(* CoDeSys 2.3 export: SOC_REAL_TO_VOLTAGE_OUT.EXP *)

(* POU SOC_real_to_Voltage_Out, ST *)
PROGRAM SOC_real_to_Voltage_Out
VAR
	TheBattery_SOC_real: REAL;
	EV_control_signal: REAL;
END_VAR
EV_control_signal := TheBattery_SOC_real/10;
END_PROGRAM
